FUNCTION TryConvert_STRING_TO_REAL : BOOL
VAR_INPUT
	in : STRING;
	out : REFERENCE TO REAL;
END_VAR

IF in <> REAL_TO_STRING(STRING_TO_REAL(in)) THEN
	RETURN;
END_IF

out := STRING_TO_REAL(in);
TryConvert_STRING_TO_REAL := TRUE;

END_FUNCTION

(* stored: Version 1.1.0.1, ProductVersion 3.1.4024.12
   POU TryConvert_STRING_TO_REAL: Id {598ad8b1-108b-4b07-be54-c75ef94a8ca1}, SpecialFunc None *)
